// TIA Portal V18 export
// export: Created 2026-01-09T11:31:56.9336949Z, ExportSetting WithDefaults, DisplayName Totally Integrated Automation Portal, DisplayVersion V18 Update 5, DisplayName TIA Portal Openness, DisplayVersion V18 Update 5, DisplayName TIA Portal Teamcenter Gateway, DisplayVersion V18, DisplayName TIA Portal Version Control Interface, DisplayVersion V18, DisplayName SINAMICS Startdrive Advanced, DisplayVersion V18 SP2 Update 1, DisplayName SINAMICS Startdrive G110M, G120, G120C, G120D, G120P, G115D, DisplayVersion V18 SP2 Update 1, DisplayName SINAMICS Startdrive G130, G150, S120, S150, SINAMICS MV, S210, G220, S200, DisplayVersion V18 SP2 Update 1, DisplayName STEP 7 Professional, DisplayVersion V18 Update 5, DisplayName STEP 7 Safety, DisplayVersion V18, DisplayName WinCC Professional, DisplayVersion V18 Update 5
TagTable "ST350_ChangeOver"
  RecipeDB_Recipe_Equal : Bool  (PLC tag ST10_RecipeDB.Recipe.Equal, CPU S71500-2PN_TP700, 1 s)
  RecipeDB_Recipe_PreConfigType : String  (PLC tag ST10_RecipeDB.Recipe.PreConfigType, CPU S71500-2PN_TP700, 1 s)
  RecipeDB_Recipe_Pulse : Bool  (PLC tag ST10_RecipeDB.Recipe.Pulse, CPU S71500-2PN_TP700, 100 ms)
    on ChangeValue: VB_RecipeST10()
  RecipeDB_Recipe_RecipeTag : String  (PLC tag ST10_RecipeDB.Recipe.RecipeTag, CPU S71500-2PN_TP700, 1 s)
  RecipeDB_Recipe_RecordName : String  (PLC tag ST10_RecipeDB.Recipe.RecordName, CPU S71500-2PN_TP700, 1 s)
  RecipeDB_Recipe_Trigger : Bool  (PLC tag ST10_RecipeDB.Recipe.Trigger, CPU S71500-2PN_TP700, 1 s)
  RecipeDB_Recipe_DataRecord_TransferStatus : Int  (PLC tag ST10_RecipeDB.Recipe.DataRecord_TransferStatus, CPU S71500-2PN_TP700, 1 s)
  Recipe_Processing_status : Int  (1 s)
